FUNCTION F_NormalizationLayer : BOOL
VAR_INPUT
	pointer_input : POINTER TO LREAL;
	pointer_mean : POINTER TO LREAL;
	pointer_std : POINTER TO LREAL;
	invert: BOOL;
	num_neurons : UINT;
END_VAR
VAR
	in : UINT;
	id : UINT;
END_VAR

IF NOT invert THEN
	FOR in := 0 TO num_neurons-1 DO
		pointer_input[in] := F_normalization(x:=pointer_input[in],mean:=pointer_mean[in],std:=pointer_std[in]);
	END_FOR
ELSE
	FOR id := 0 TO num_neurons-1 DO
		 pointer_input[id] := F_denormalization(x:=pointer_input[id],mean:=pointer_mean[id],std:=pointer_std[id]);
	END_FOR
END_IF

END_FUNCTION

(* stored: Version 1.1.0.1, ProductVersion 3.1.4024.12
   POU F_NormalizationLayer: Id {f60f2a43-f25f-4ac3-8998-e7bbd7e457a7}, SpecialFunc None *)
